VAR_GLOBAL CONSTANT
	cintMaxDecisions: INT := 300;
END_VAR

(* stored: Version 1.1.0.1, ProductVersion 3.1.0.19
   GVL Const_DPJ: Id {7c6d5798-41ef-44f0-ba5e-daf571ec2692} *)
